// TIA Portal V16 export
// export: Created 2022-11-17T11:57:52.7701562Z, ExportSetting WithDefaults, DisplayName Totally Integrated Automation Portal, DisplayVersion V16 Update 6, DisplayName TIA Portal Version Control Interface, DisplayVersion V16 Update 2, DisplayName TIA Portal Openness, DisplayVersion V16 Update 6, DisplayName SINAMICS Startdrive Advanced, DisplayVersion V16 Update 5, DisplayName SINAMICS Startdrive G130, G150, S120, S150, SINAMICS MV, S210, DisplayVersion V16 Update 5, DisplayName SINAMICS Startdrive G110M, G120, G120C, G120D, G120P, G115D, DisplayVersion V16 Update 5, DisplayName STEP 7 Professional, DisplayVersion V16 Update 6, DisplayName STEP 7 Safety, DisplayVersion V16, DisplayName WinCC Advanced, DisplayVersion V16 Update 6
DATA_BLOCK "SINA_SPEED_Motor_Centrador_DB"   // DB11
AUTHOR : DRVDPS7
FAMILY : DRIVES
NAME : SINA_SPD
VERSION : 5.1
// stored: AutoNumber true, InstanceOfName SINA_SPEED_Motor_Centrador, InstanceOfType FB
"SINA_SPEED_Motor_Centrador"
   // VAR_INPUT
   //    EnableAxis : Bool;
   //    AckError : Bool;
   //    SpeedSp : Real;
   //    RefSpeed : Real;
   //    ConfigAxis : Word;
   //    HWIDSTW : HW_IO;
   //    HWIDZSW : HW_IO;
   // END_VAR
   // VAR_OUTPUT
   //    AxisEnabled : Bool;
   //    Lockout : Bool;
   //    ActVelocity : Real;
   //    Error : Bool;
   //    Status : Word;
   //    DiagId : Word;
   // END_VAR
   // VAR
   //    sxSendBuf : Struct
   //       STW1 : Word;
   //       Velocity : Word;
   //    END_STRUCT;
   //    sxRecvBuf : Struct
   //       ZSW1 : Word;
   //       Velocity : Word;
   //    END_STRUCT;
   // END_VAR
BEGIN
END_DATA_BLOCK
